TYPE "tAutoShipping"
VERSION : 0.8
   STRUCT
      "standard" : "tAutoStandard";
      index : "tIndex";
   END_STRUCT;

END_TYPE

